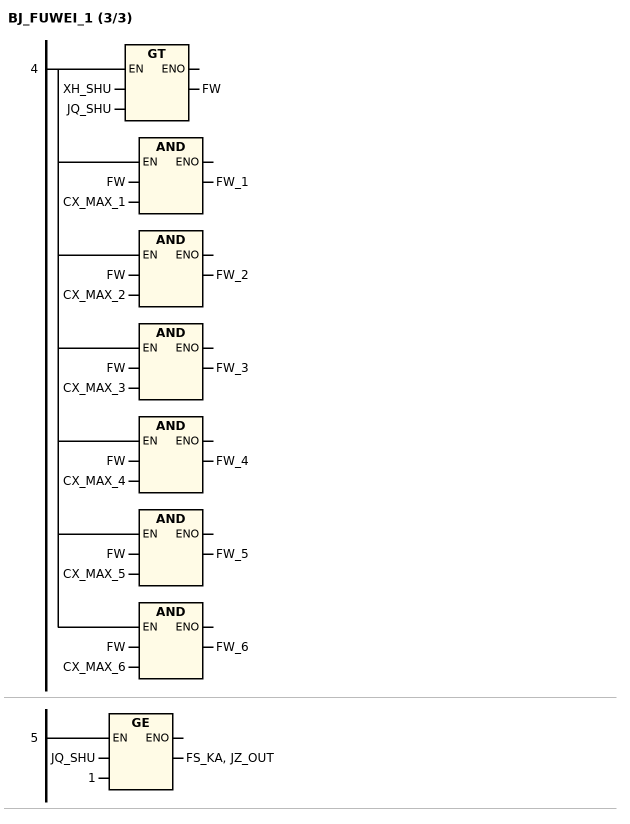
[picture p120: BJ_FUWEI_1 (LD)]
_LD_ (* Ladder Diagram *)
NETWORK 1
	*
		EN --- ADD(BOOL_TO_WORD(GE(XH_SHUI, 3)), BOOL_TO_WORD(GE(XH_SHUI, 6)), BOOL_TO_WORD(GE(XH_SHUI, 9)), BOOL_TO_WORD(GE(XH_SHUI, 12)), BOOL_TO_WORD(GE(XH_SHUI, 15)), BOOL_TO_WORD(GE(XH_SHUI, 18))) => XH_SHU
NETWORK 2
	*
		EN --- ADD(BOOL_TO_WORD(JQ_1), BOOL_TO_WORD(JQ_2), BOOL_TO_WORD(JQ_3), BOOL_TO_WORD(JQ_4), BOOL_TO_WORD(JQ_5), BOOL_TO_WORD(JQ_6)) => JQ_SHU
NETWORK 3
	*
		EN --- MAX(MAX(MAX(MAX(MAX(SEL(AND(EQ(CX_1_1, 0), NOT EQ(CX_1_1, CX_1), NOT CHD_1), 0, CX_1), SEL(AND(EQ(CX_2_1, 0), NOT EQ(CX_2_1, CX_2), NOT CHD_2), 0, CX_2)), SEL(AND(EQ(CX_3_1, 0), NOT EQ(CX_3_1, CX_3), NOT CHD_3), 0, CX_3)), SEL(AND(EQ(CX_4_1, 0), NOT EQ(CX_4_1, CX_4), NOT CHD_4), 0, CX_4)), SEL(AND(EQ(CX_5_1, 0), NOT EQ(CX_5_1, CX_5), NOT CHD_5), 0, CX_5)), SEL(AND(EQ(CX_6_1, 0), NOT EQ(CX_6_1, CX_6), NOT CHD_6), 0, CX_6)) => CX_MAX1
		EN --- EQ(CX_MAX1, CX_1) => CX_MAX_1
		EN --- EQ(CX_MAX1, CX_2) => CX_MAX_2
		EN --- EQ(CX_MAX1, CX_3) => CX_MAX_3
		EN --- EQ(CX_MAX1, CX_4) => CX_MAX_4
		EN --- EQ(CX_MAX1, CX_5) => CX_MAX_5
		EN --- EQ(CX_MAX1, CX_6) => CX_MAX_6
NETWORK 4
	*
		EN --- GT(XH_SHU, JQ_SHU) => FW
		EN --- AND(FW, CX_MAX_1) => FW_1
		EN --- AND(FW, CX_MAX_2) => FW_2
		EN --- AND(FW, CX_MAX_3) => FW_3
		EN --- AND(FW, CX_MAX_4) => FW_4
		EN --- AND(FW, CX_MAX_5) => FW_5
		EN --- AND(FW, CX_MAX_6) => FW_6
NETWORK 5
	*
		EN --- GE(JQ_SHU, 1) => FS_KA, JZ_OUT
_END_LD_
(* the same logic as Structured Text *)
(* Network 1 *)
XH_SHU := BOOL_TO_WORD(XH_SHUI >= 3) + BOOL_TO_WORD(XH_SHUI >= 6) + BOOL_TO_WORD(XH_SHUI >= 9) + BOOL_TO_WORD(XH_SHUI >= 12) + BOOL_TO_WORD(XH_SHUI >= 15) + BOOL_TO_WORD(XH_SHUI >= 18);
(* Network 2 *)
JQ_SHU := BOOL_TO_WORD(JQ_1) + BOOL_TO_WORD(JQ_2) + BOOL_TO_WORD(JQ_3) + BOOL_TO_WORD(JQ_4) + BOOL_TO_WORD(JQ_5) + BOOL_TO_WORD(JQ_6);
(* Network 3 *)
CX_MAX1 := MAX(MAX(MAX(MAX(MAX(SEL((CX_1_1 = 0) AND NOT (CX_1_1 = CX_1) AND NOT CHD_1, 0, CX_1), SEL((CX_2_1 = 0) AND NOT (CX_2_1 = CX_2) AND NOT CHD_2, 0, CX_2)), SEL((CX_3_1 = 0) AND NOT (CX_3_1 = CX_3) AND NOT CHD_3, 0, CX_3)), SEL((CX_4_1 = 0) AND NOT (CX_4_1 = CX_4) AND NOT CHD_4, 0, CX_4)), SEL((CX_5_1 = 0) AND NOT (CX_5_1 = CX_5) AND NOT CHD_5, 0, CX_5)), SEL((CX_6_1 = 0) AND NOT (CX_6_1 = CX_6) AND NOT CHD_6, 0, CX_6));
CX_MAX_1 := CX_MAX1 = CX_1;
CX_MAX_2 := CX_MAX1 = CX_2;
CX_MAX_3 := CX_MAX1 = CX_3;
CX_MAX_4 := CX_MAX1 = CX_4;
CX_MAX_5 := CX_MAX1 = CX_5;
CX_MAX_6 := CX_MAX1 = CX_6;
(* Network 4 *)
FW := XH_SHU > JQ_SHU;
FW_1 := FW AND CX_MAX_1;
FW_2 := FW AND CX_MAX_2;
FW_3 := FW AND CX_MAX_3;
FW_4 := FW AND CX_MAX_4;
FW_5 := FW AND CX_MAX_5;
FW_6 := FW AND CX_MAX_6;
(* Network 5: see the listing above *)
END_FUNCTION_BLOCK

(* POU WD_XH, LD *)
FUNCTION_BLOCK WD_XH
VAR
	PJ_ANNIU: AN_NIU;

	DCF_OFF: BOOL;

END_VAR
VAR_INPUT
	WD_1_IN: INT;
	WD_2_IN: INT;
	WD_3_IN: INT;


	PJ_IN: BOOL;
	TT_SHU: WORD;


END_VAR
VAR_OUTPUT

	PJ_OUT: BOOL;
	KF_WD_OUT: INT;

END_VAR
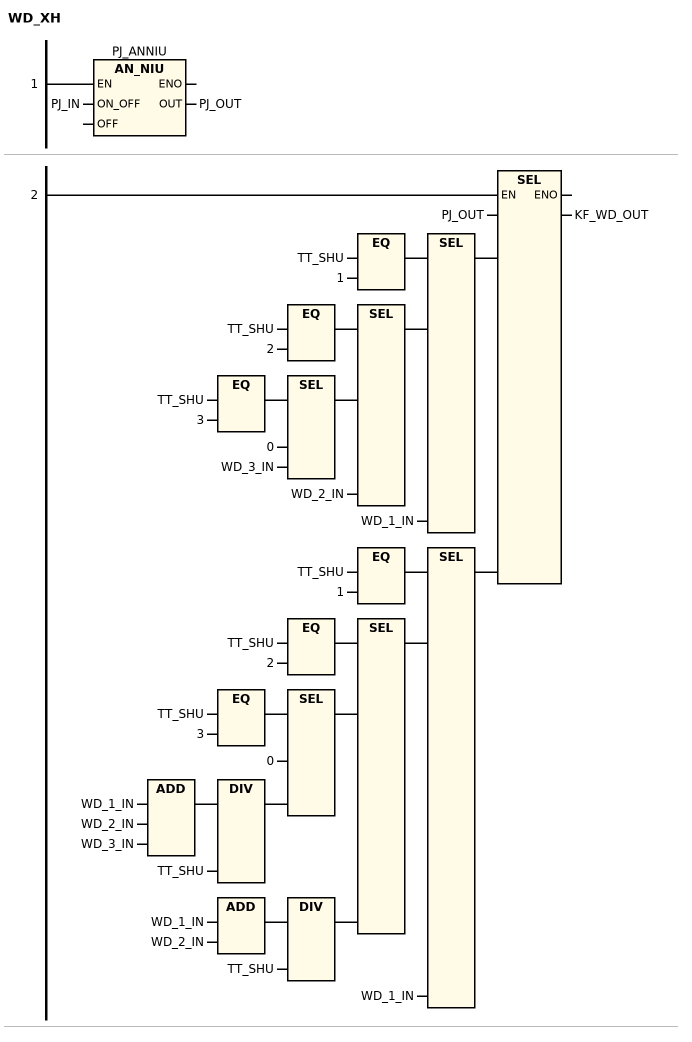
_LD_ (* Ladder Diagram *)
NETWORK 1
	*
		EN --- PJ_ANNIU:AN_NIU(ON_OFF: PJ_IN, OFF: ) => PJ_OUT
NETWORK 2
	*
		EN --- SEL(PJ_OUT, SEL(EQ(TT_SHU, 1), SEL(EQ(TT_SHU, 2), SEL(EQ(TT_SHU, 3), 0, WD_3_IN), WD_2_IN), WD_1_IN), SEL(EQ(TT_SHU, 1), SEL(EQ(TT_SHU, 2), SEL(EQ(TT_SHU, 3), 0, DIV(ADD(WD_1_IN, WD_2_IN, WD_3_IN), TT_SHU)), DIV(ADD(WD_1_IN, WD_2_IN), TT_SHU)), WD_1_IN)) => KF_WD_OUT
_END_LD_
(* the same logic as Structured Text *)
(* Network 1: see the listing above *)
(* Network 2 *)
KF_WD_OUT := SEL(PJ_OUT, SEL(TT_SHU = 1, SEL(TT_SHU = 2, SEL(TT_SHU = 3, 0, WD_3_IN), WD_2_IN), WD_1_IN), SEL(TT_SHU = 1, SEL(TT_SHU = 2, SEL(TT_SHU = 3, 0, (WD_1_IN + WD_2_IN + WD_3_IN) / TT_SHU), (WD_1_IN + WD_2_IN) / TT_SHU), WD_1_IN));
END_FUNCTION_BLOCK

(* POU BB, LD *)
FUNCTION_BLOCK BB
VAR_INPUT
	JZ_IN: BOOL;
	ZQ_IN: WORD;
	BJ_IN: BOOL;
END_VAR
VAR_OUTPUT
	CF_OUT: BOOL;
END_VAR
VAR
	BLINK: BLINK;
	R_TRIG: R_TRIG;
	TOF: TOF;
	TOF1: TOF;
	F_TRIG: F_TRIG;
	R_TRI2: R_TRIG;
	TOF2: TOF;
END_VAR
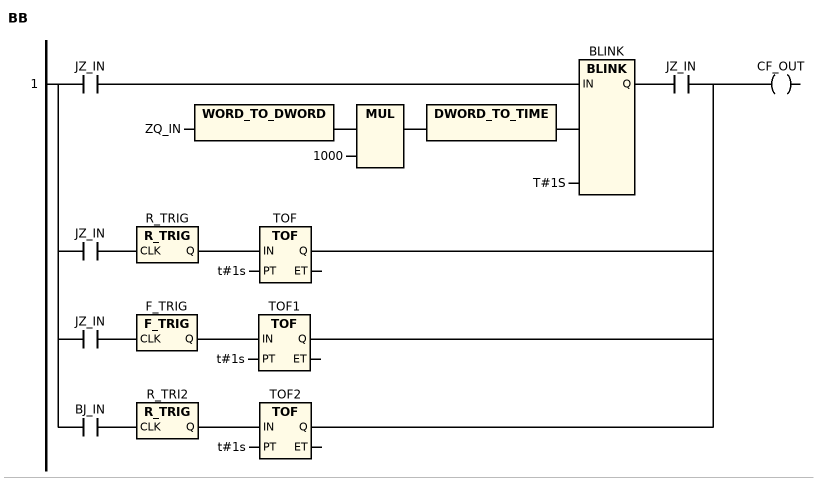
_LD_ (* Ladder Diagram *)
NETWORK 1
	{ [JZ_IN] - BLINK:BLINK(*, DWORD_TO_TIME(MUL(WORD_TO_DWORD(ZQ_IN), 1000)), T#1S) - [JZ_IN] | [JZ_IN] - R_TRIG:R_TRIG(CLK: *) - TOF:TOF(IN: *, PT: t#1s) | [JZ_IN] - F_TRIG:F_TRIG(CLK: *) - TOF1:TOF(IN: *, PT: t#1s) | [BJ_IN] - R_TRI2:R_TRIG(CLK: *) - TOF2:TOF(IN: *, PT: t#1s) } --- (CF_OUT)
_END_LD_
END_FUNCTION_BLOCK
